(* PLC project cmd_double_acting_jack, Dassault Systèmes ControlBuild 2024x *)
(* stored: creationDateTime 2023-10-03T11:13:35-01:00 *)

FUNCTION_BLOCK actuator
  VAR_INPUT
    autoMode : BOOL := false;
    manualMode : BOOL := false;
  END_VAR
  VAR_INPUT
    autoWorkCmd : BOOL := false;
    autoRestCmd : BOOL := false;
  END_VAR
  VAR_INPUT
    valveWorkPB : BOOL := false;
    valveRestPB : BOOL := false;
  END_VAR
  VAR_INPUT
    outletSensor : BOOL := false;
    inletSensor : BOOL := false;
  END_VAR
  VAR_INPUT
    generalFault : BOOL := false;
  END_VAR
  VAR_OUTPUT
    workCmd : BOOL := false;
    restCmd : BOOL := false;
  END_VAR

(* LD diagram, written out as Structured Text *)
1:
workCmd := (autoMode AND (autoWorkCmd OR workCmd) AND NOT autoRestCmd OR manualMode AND valveWorkPB AND NOT valveRestPB OR manualMode AND workCmd) AND NOT outletSensor AND NOT generalFault;
2:
restCmd := (autoMode AND (autoRestCmd OR restCmd) AND NOT autoWorkCmd OR manualMode AND valveRestPB AND NOT valveWorkPB OR manualMode AND restCmd) AND NOT inletSensor AND NOT generalFault;
END_FUNCTION_BLOCK

FUNCTION_BLOCK faults
  VAR_INPUT
    workCmd : BOOL := false;
    restCmd : BOOL := false;
  END_VAR
  VAR_INPUT
    outletSensor : BOOL := false;
    inletSensor : BOOL := false;
  END_VAR
  VAR_INPUT
    acknowledgePB : BOOL := false;
  END_VAR
  VAR_OUTPUT
    generalFault : BOOL := false;
  END_VAR
  VAR
    discordanceFault : BOOL := false;
    outletSensorFault : BOOL := false;
    inletSensorFault : BOOL := false;
  END_VAR
  VAR CONSTANT
    presetMvt : TIME := T#0h0m10s0ms;
    presetDiscordance : TIME := T#0h0m0s200ms;
  END_VAR

(* LD diagram, written out as Structured Text *)
1:
IF acknowledgePB THEN discordanceFault := FALSE; END_IF;
IF acknowledgePB THEN outletSensorFault := FALSE; END_IF;
IF acknowledgePB THEN inletSensorFault := FALSE; END_IF;
IF acknowledgePB THEN generalFault := FALSE; END_IF;
2:
TON_OUT(IN := workCmd, PT := presetMvt);
IF TON_OUT.Q0 AND NOT outletSensor THEN outletSensorFault := TRUE; END_IF;
TON_IN(IN := restCmd, PT := presetMvt);
IF TON_IN.Q0 AND NOT inletSensor THEN inletSensorFault := TRUE; END_IF;
3:
TON_DISC(IN := outletSensor AND inletSensor, PT := presetDiscordance);
IF TON_DISC.Q0 THEN discordanceFault := TRUE; END_IF;
4:
IF discordanceFault OR outletSensorFault OR inletSensorFault THEN generalFault := TRUE; END_IF;
END_FUNCTION_BLOCK

(* Command of a double acting jack with fault detection *)
PROGRAM cmd_equipment_library.cmd_double_acting_jack
  VAR_INPUT
    autoMode : BOOL := false;
    manualMode : BOOL := false;
  END_VAR
  VAR_INPUT
    autoWorkCmd : BOOL := false;
    autoRestCmd : BOOL := false;
  END_VAR
  VAR_INPUT
    valveWorkPB : BOOL := false;
    valveRestPB : BOOL := false;
  END_VAR
  VAR_INPUT
    outletSensor : BOOL := false;
    inletSensor : BOOL := false;
  END_VAR
  VAR_INPUT
    acknowledgePB : BOOL := false;
  END_VAR
  VAR_OUTPUT
    workCmd : BOOL := false;
    restCmd : BOOL := false;
  END_VAR
  VAR_OUTPUT
    generalFault : BOOL := false;
  END_VAR

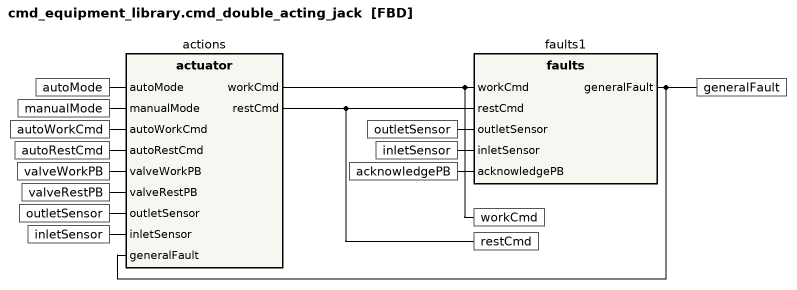
(* FBD diagram, written out as Structured Text *)
faults1(workCmd := actions.workCmd, restCmd := actions.restCmd, outletSensor := outletSensor, inletSensor := inletSensor, acknowledgePB := acknowledgePB);
actions(autoMode := autoMode, manualMode := manualMode, autoWorkCmd := autoWorkCmd, autoRestCmd := autoRestCmd, valveWorkPB := valveWorkPB, valveRestPB := valveRestPB, outletSensor := outletSensor, inletSensor := inletSensor, generalFault := faults1.generalFault);
workCmd := actions.workCmd;
restCmd := actions.restCmd;
generalFault := faults1.generalFault;
END_PROGRAM
